{attribute addProperty BoxType "EK1122-0000-0018"}
{attribute addProperty Id "Beckhoff_BKxxxxsub_EK1100Beckhoff_BKxxxxsub_EK1100_CE1F492600A_0001_BK1120_0000_0000A_0001_BK1120_0000_0000_A11D37A600A_0002_BK1120_0000_0001A_0002_BK1120_0000_0001_6C91631300A_0003_BK1120_0000_0016A_0003_BK1120_0000_0016_3EC4837B00A_0004_BK1120_0000_0017A_0004_BK1120_0000_0017_F348D7CE00A_0005_BK1120_0000_0018A_0005_BK1120_0000_0018_EC8BABB100A_0006_BK1120_0000_0019A_0006_BK1120_0000_0019_2107FF0400A_0007_BK1120_0000_0020A_0007_BK1120_0000_0020_2D4D5A6600A_0008_BK1120_0000_0021A_0008_BK1120_0000_0021_E0C10ED300A_0009_CPXXXX_BK1150_0016A_0009_CPXXXX_BK1150_0016_B294EEBB00A_0010_BK1150_0000_0016A_0010_BK1150_0000_0016_7F18BA0E00A_0011_BK1150_0000_0017A_0011_BK1150_0000_0017_163F2E6B00A_0012_BK1150_0000_0018A_0012_BK1150_0000_0018_DBB37ADE00A_0013_BK1150_0000_0019A_0013_BK1150_0000_0019_89E69AB600Term_474_EK1100Term_474_EK1100_44DC070B00Term_476_EK1100Term_476_EK1100_ED4AD6ED00Term_478_EK1100Term_478_EK1100_69E708A200A_0019_IL2300_B110_0016A_0019_IL2300_B110_0016_D7C567E600A_0020_IL2300_B110_0017A_0020_IL2300_B110_0017_5C3C5D5200A_0021_IL2301_B110_0016A_0021_IL2301_B110_0016_18E5DAA800A_0022_IL2301_B110_0017A_0022_IL2301_B110_0017_CE2B414F00A_0023_IL2302_B110_0016A_0023_IL2302_B110_0016_9156D55C00A_0024_IL2302_B110_0017A_0024_IL2302_B110_0017_7CD378DF00"}
{attribute addProperty CRC "4074462217"}
{attribute addProperty SizeInBites "0"}
{attribute addProperty SizeInBytes "0"}
TYPE Beckhoff_BKxxxxEK1122_F2DB5C09 EXTENDS EK1122_179A0949 :
STRUCT
	{attribute addProperty Name "Beckhoff_BKxxxxsub_EK1100"}
	Beckhoff_BKxxxxsub_EK1100 : Beckhoff_BKxxxxsub_EK1100_CE1F4926;
	{attribute addProperty Name "A_0001_BK1120_0000_0000"}
	A_0001_BK1120_0000_0000 : A_0001_BK1120_0000_0000_A11D37A6;
	{attribute addProperty Name "A_0002_BK1120_0000_0001"}
	A_0002_BK1120_0000_0001 : A_0002_BK1120_0000_0001_6C916313;
	{attribute addProperty Name "A_0003_BK1120_0000_0016"}
	A_0003_BK1120_0000_0016 : A_0003_BK1120_0000_0016_3EC4837B;
	{attribute addProperty Name "A_0004_BK1120_0000_0017"}
	A_0004_BK1120_0000_0017 : A_0004_BK1120_0000_0017_F348D7CE;
	{attribute addProperty Name "A_0005_BK1120_0000_0018"}
	A_0005_BK1120_0000_0018 : A_0005_BK1120_0000_0018_EC8BABB1;
	{attribute addProperty Name "A_0006_BK1120_0000_0019"}
	A_0006_BK1120_0000_0019 : A_0006_BK1120_0000_0019_2107FF04;
	{attribute addProperty Name "A_0007_BK1120_0000_0020"}
	A_0007_BK1120_0000_0020 : A_0007_BK1120_0000_0020_2D4D5A66;
	{attribute addProperty Name "A_0008_BK1120_0000_0021"}
	A_0008_BK1120_0000_0021 : A_0008_BK1120_0000_0021_E0C10ED3;
	{attribute addProperty Name "A_0009_CPXXXX_BK1150_0016"}
	A_0009_CPXXXX_BK1150_0016 : A_0009_CPXXXX_BK1150_0016_B294EEBB;
	{attribute addProperty Name "A_0010_BK1150_0000_0016"}
	A_0010_BK1150_0000_0016 : A_0010_BK1150_0000_0016_7F18BA0E;
	{attribute addProperty Name "A_0011_BK1150_0000_0017"}
	A_0011_BK1150_0000_0017 : A_0011_BK1150_0000_0017_163F2E6B;
	{attribute addProperty Name "A_0012_BK1150_0000_0018"}
	A_0012_BK1150_0000_0018 : A_0012_BK1150_0000_0018_DBB37ADE;
	{attribute addProperty Name "A_0013_BK1150_0000_0019"}
	A_0013_BK1150_0000_0019 : A_0013_BK1150_0000_0019_89E69AB6;
	{attribute addProperty Name "Term_474_EK1100"}
	Term_474_EK1100 : Term_474_EK1100_44DC070B;
	{attribute addProperty Name "Term_476_EK1100"}
	Term_476_EK1100 : Term_476_EK1100_ED4AD6ED;
	{attribute addProperty Name "Term_478_EK1100"}
	Term_478_EK1100 : Term_478_EK1100_69E708A2;
	{attribute addProperty Name "A_0019_IL2300_B110_0016"}
	A_0019_IL2300_B110_0016 : A_0019_IL2300_B110_0016_D7C567E6;
	{attribute addProperty Name "A_0020_IL2300_B110_0017"}
	A_0020_IL2300_B110_0017 : A_0020_IL2300_B110_0017_5C3C5D52;
	{attribute addProperty Name "A_0021_IL2301_B110_0016"}
	A_0021_IL2301_B110_0016 : A_0021_IL2301_B110_0016_18E5DAA8;
	{attribute addProperty Name "A_0022_IL2301_B110_0017"}
	A_0022_IL2301_B110_0017 : A_0022_IL2301_B110_0017_CE2B414F;
	{attribute addProperty Name "A_0023_IL2302_B110_0016"}
	A_0023_IL2302_B110_0016 : A_0023_IL2302_B110_0016_9156D55C;
	{attribute addProperty Name "A_0024_IL2302_B110_0017"}
	A_0024_IL2302_B110_0017 : A_0024_IL2302_B110_0017_7CD378DF;
END_STRUCT
END_TYPE

(* stored: Version 1.2.0.0, ProductVersion 3.1.4024.9
   DUT Beckhoff_BKxxxxEK1122_F2DB5C09: Id {03146bae-40f9-4ae0-bf5d-8364dd050d56} *)
